Fanuc KAREL source: graph.kl

PROGRAM graph
%NOBUSYLAMP
%COMMENT = 'graph routines'
%NOLOCKGROUP
%NOPAUSE = COMMAND + TPENABLE + ERROR

%include systemlib.klt

%include graph.klt

%include graph_algo.private.klh
%include graph_algo.klh


--private

--public

BEGIN
END graph
